{attribute 'GeneratedUsingTerminal: IODEVICETYPE_ETHERCATPROT'}
{attribute addProperty BoxType "IODEVICETYPE_ETHERCATPROT"}
{attribute addProperty Id "Beckhoff_EP1xxxBeckhoff_EP1xxx_6D0137A81740Beckhoff_EP2xxxBeckhoff_EP2xxx_E245E7283524Beckhoff_EP3xxxBeckhoff_EP3xxx_375966123196Beckhoff_EP4xxxBeckhoff_EP4xxx_3C0BABAE336Beckhoff_EP5xxxBeckhoff_EP5xxx_6BDCDC3F409Beckhoff_EP6xxxBeckhoff_EP6xxx_E108946E1410Beckhoff_EP7xxxBeckhoff_EP7xxx_7139B48E2992Beckhoff_EP8xxxBeckhoff_EP8xxx_EBB5A763282Beckhoff_EP9xxxBeckhoff_EP9xxx_33F6D646617SyncUnitsSyncUnits_2E61B95536InputsInputs_25A0042B160OutputsOutputs_2397A10E106InfoDataInfoData_E68C61CD28"}
{attribute addProperty CRC "1016939505"}
{attribute addProperty Size "14836"}
TYPE EtherCAT_Master_EPxxxx_3C9D43F1 :
STRUCT
	{attribute addProperty Name "Beckhoff_EP1xxx"}
	Beckhoff_EP1xxx : Beckhoff_EP1xxx_6D0137A8;
	{attribute addProperty Name "Beckhoff_EP2xxx"}
	Beckhoff_EP2xxx : Beckhoff_EP2xxx_E245E728;
	{attribute addProperty Name "Beckhoff_EP3xxx"}
	Beckhoff_EP3xxx : Beckhoff_EP3xxx_37596612;
	{attribute addProperty Name "Beckhoff_EP4xxx"}
	Beckhoff_EP4xxx : Beckhoff_EP4xxx_3C0BABAE;
	{attribute addProperty Name "Beckhoff_EP5xxx"}
	Beckhoff_EP5xxx : Beckhoff_EP5xxx_6BDCDC3F;
	{attribute addProperty Name "Beckhoff_EP6xxx"}
	Beckhoff_EP6xxx : Beckhoff_EP6xxx_E108946E;
	{attribute addProperty Name "Beckhoff_EP7xxx"}
	Beckhoff_EP7xxx : Beckhoff_EP7xxx_7139B48E;
	{attribute addProperty Name "Beckhoff_EP8xxx"}
	Beckhoff_EP8xxx : Beckhoff_EP8xxx_EBB5A763;
	{attribute addProperty Name "Beckhoff_EP9xxx"}
	Beckhoff_EP9xxx : Beckhoff_EP9xxx_33F6D646;
	{attribute addProperty Name "SyncUnits"}
	SyncUnits : SyncUnits_2E61B955;
	{attribute addProperty Name "Inputs"}
	Inputs : Inputs_25A0042B;
	{attribute addProperty Name "Outputs"}
	Outputs : Outputs_2397A10E;
	{attribute addProperty Name "InfoData"}
	InfoData : InfoData_E68C61CD;
END_STRUCT
END_TYPE

(* stored: Version 1.2.0.0, ProductVersion 3.1.4024.9
   DUT EtherCAT_Master_EPxxxx_3C9D43F1: Id {9e2e0e88-6cc9-48bc-b694-97cc4baf8b88} *)
